TEXTLIST ErrorList
  0 = 'Minden rendben.'
  1 = 'Termék csatlakozó fedél\nnincs nyitva.'
  2 = 'Termék csatlakozó fedél\nnyitva van.'
  3 = 'Fütötömb hömérséklete\nnem megfelelö.'
  4 = 'Fütötömb hömérséklete\nmegfelelö.'
  5 = 'Sürített levegö nyomása\nnincs rendben.'
  6 = 'Sürített levegö nem kapcsolt ki.'
  7 = 'Nincs hegesztö\nelöfigyelmeztetés.'
  8 = 'Hegesztö\nelöfigyelmeztetés!'
  9 = 'Nem kell hegesztö elektródát\ncserélni.'
  10 = 'Hegesztö elektródát\nkell cserélni.'
  11 = 'A hegesztö még nem\nindult be.'
  12 = 'A hegesztö beindult.'
  13 = 'Nincs hegesztö áramhiba.'
  14 = 'Hegesztö áramhiba!'
  15 = 'Árammal hegesztés\nkikapcsolva!'
  16 = 'Árammal hegesztés\nbekapcsolva!'
  17 = 'A hegesztö nem üzemkész!'
  18 = 'A hegesztö üzemkész!'
  19 = 'NTC vágó: sebesség\nnem nulla.'
  20 = 'NTC vágó: sebesség nulla.'
  21 = 'NTC vágó: a sebesség\nnem állt be!'
  22 = 'NTC vágó: a sebesség\nbeállt!'
  23 = 'NTC vágó: nincs vészjelzés.'
  24 = 'NTC vágó: vészjelzés!'
  25 = 'NTC vágó: nem üzemkész!'
  26 = 'NTC vágó: üzemkész.'
  27 = 'Hegesztö: hegesztési\nfolyamat nincs kész.'
  28 = 'Hegesztö: hegesztési\nfolyamat kész.'
  29 = 'Pt oldali fénysorompó\nblokkolva.'
  30 = 'Pt oldali fénysorompó\nszabad.'
  31 = 'NTC oldali fénysorompó\nblokkolva.'
  32 = 'NTC oldali fénysorompó\nszabad.'
  33 = 'A kamera dolgozik.'
  34 = 'A kamera nem dolgozik.'
  35 = 'Kamera: a termék nincs jól\nrögzitve.'
  36 = 'Kamera: a termék jól\nvan rögzitve.'
  37 = 'Kamera: vezeték színsorrend\nnincs rendben.'
  38 = 'Kamera: vezeték színsorrend\nrendben van.'
  39 = 'Kamera: vezeték szigetelés\nnincs rendben.'
  40 = 'Kamera: vezeték szigetelés\nrendben van.'
  41 = 'A biztonsági relé földje megvan.'
  42 = 'A biztonsági relé földje hiányzik.\nValamelyik ajtó nyitva van?'
  43 = 'A biztonsági relé tápja hiányzik.\nValamelyik ajtó nyitva van?'
  44 = 'A biztonsági relé tápja megvan.'
  65 = 'Adapterlefogó nincs\nteljesen visszahúzva.'
  66 = 'Adapterlefogó\nteljesen visszahúzva.'
  67 = 'Adapterlefogó nem\naktiválódott.'
  68 = 'Az adapterlefogó aktív.'
  69 = 'Nem érzékel adaptert\na szánon!'
  70 = 'Fent van az adapter a szánon.'
  71 = 'A 3-as hegesztöfej nincs fent.'
  72 = 'A 3-as hegesztöfej fent van.'
  73 = 'A 3-as hegesztöfej nincs lent.'
  74 = 'A 3-as hegesztöfej lent van.'
  75 = 'A Pt oldali tengely plusz\nvégállásban van.'
  76 = 'A Pt oldali tengely nincs\nplusz \nvégállásban.'
  81 = 'Fütötömb nincs fent.'
  82 = 'Fütötömb fent van.'
  83 = 'Fütötömb nincs lent.'
  84 = 'Fütötömb lent van.'
  85 = 'Mérötük nincsenek kitolva.'
  86 = 'Mérötük ki vannak tolva.'
  87 = 'Mérötük nincsenek behúzva.'
  88 = 'Mérötük be vannak húzva.'
  89 = 'Lézer blende nincs bezárva.'
  90 = 'Lézer blende be van zárva.'
  91 = 'Lézer blende nincs kinyitva.'
  92 = 'Lézer blende ki van nyitva.'
  93 = 'Kappe prés legalul van.'
  94 = 'Kappe prés nincs legalul.'
  95 = 'A Pt oldali tengely minusz\nvégállásban van.'
  96 = 'A Pt oldali tengely nincs\nminusz \nvégállásban.'
  97 = 'Kappe prés jobb oldala\nnincs lent.'
  98 = 'Kappe prés jobb oldala\nlent van.'
  99 = 'Kappe prés jobb oldala\nnincs fent.'
  100 = 'Kappe prés jobb oldala\nfent van.'
  101 = 'Kappe prés bal oldala\nnincs fent.'
  102 = 'Kappe prés bal oldala\nfent van.'
  103 = 'Kappe prés bal oldala\nnincs lent.'
  104 = 'Kappe prés bal oldala\nlent van.'
  105 = 'A fütötömb nincs a szán\nfölött.'
  106 = 'A fütötömb a szán \nfölött van.'
  107 = 'A szigetelés mérötük\nnincsenek a szán fölött.'
  108 = 'A szigetelés mérötük\na szán fölött vannak.'
  109 = 'A kappe prés nincs fent.'
  110 = 'A kappe prés fent van.'
  111 = 'A nagyfeszültségü mérötü\nnincs lent.'
  112 = 'A nagyfeszültségü mérötü\nlent van.'
  113 = 'NTC vágó: vágó-hajlító\nnincs lent.'
  114 = 'NTC vágó: vágó-hajlító\nlent van.'
  115 = 'NTC vágó: vágó-hajlító\nnincs fent.'
  116 = 'NTC vágó: vágó-hajlító\nfent van.'
  117 = '2. hegesztö fej: Felsö elektróda\nnincs kitolva.'
  118 = '2. hegesztö fej: Felsö elektróda\nki van tolva.'
  119 = '2. hegesztö fej: Felsö elektróda\nnincs behúzva.'
  120 = '2. hegesztö fej: Felsö elektróda\nbe van húzva.'
  121 = '2. hegesztö fej: Alsó elektróda\nnincs behúzva.'
  122 = '2. hegesztö fej: Alsó elektróda\nbe van húzva.'
  123 = '2. hegesztö fej: Alsó elektróda\nnincs kitolva.'
  124 = '2. hegesztö fej: Alsó elektróda\nki van tolva.'
  125 = 'NTC oldali tengely minusz\nvégállásban van.'
  126 = 'NTC oldali tengely nincs\nminusz \nvégállásban.'
  127 = 'NTC vágó: az NTC nincs\nmegfelelö pozícióban.'
  128 = 'NTC vágó: az NTC\nmegfelelö pozícióban van.'
  129 = 'NTC vágó: NTC megfogó\nnincs nyitva.'
  130 = 'NTC vágó: NTC megfogó\nnyitva van.'
  131 = 'NTC vágó: NTC megfogó\nnincs zárva.'
  132 = 'NTC vágó: NTC megfogó\nzárva van.'
  133 = 'NTC vágó: NTC kiszedö\nnincs kitolva.'
  134 = 'NTC vágó: NTC kiszedö\nki van tolva.'
  135 = 'NTC vágó: NTC kiszedö\nnincs behúzva.'
  136 = 'NTC vágó: NTC kiszedö\nbe van húzva.'
  137 = 'NTC vágó: piros gomb\nnincs benyomva.'
  138 = 'NTC vágó: piros gomb\nbe van nyomva.'
  139 = 'NTC vágó: zöld gomb\nnincs benyomva.'
  140 = 'NTC vágó: zöld gomb\nbe van nyomva.'
  141 = 'Nincs megfelelö vágott NTC.'
  142 = 'Van vágott NTC.'
  145 = 'Elöhajlító: felsö pofa nincs lent.'
  146 = 'Elöhajlító: felsö pofa lent van.'
  147 = 'Elöhajlító: felsö pofa nincs fent.'
  148 = 'Elöhajlító: felsö pofa fent van.'
  149 = 'Elöhajlító: alsó pofa nincs lent.'
  150 = 'Elöhajlító: alsó pofa lent van.'
  151 = 'Elöhajlító: alsó pofa nincs fent.'
  152 = 'Elöhajlító: alsó pofa fent van.'
  153 = '1. hegesztöfej: bal elektróda\nnincs fent.'
  154 = '1. hegesztöfej: bal elektróda\nfent van.'
  155 = '1. hegesztöfej: bal elektróda\nnincs lent.'
  156 = '1. hegesztöfej: bal elektróda\nlent van.'
  161 = 'Véghajlító: felsö pofa nincs lent.'
  162 = 'Véghajlító: felsö pofa lent van.'
  163 = 'Véghajlító: felsö pofa nincs fent.'
  164 = 'Véghajlító: felsö pofa fent van.'
  165 = 'Véghajlító: alsó pofa nincs fent.'
  166 = 'Véghajlító: alsó pofa fent van.'
  167 = 'Véghajlító: alsó pofa nincs lent.'
  168 = 'Elöhajlító: alsó pofa lent van.'
  169 = '1. hegesztöfej: jobb elektróda\nnincs fent.'
  170 = '1. hegesztöfej: jobb elektróda\nfent van.'
  171 = '1. hegesztöfej: jobb elektróda\nnincs lent.'
  172 = '1. hegesztöfej: jobb elektróda\nlent van.'
  175 = 'NTC oldali tengely plusz\nvégállásban van.'
  176 = 'NTC oldali tengely nincs\nplusz végállásban.'
  193 = 'NTC oldali tengely nem\nüzemkész.'
  194 = 'NTC oldali tengely\nüzemkész.'
  195 = 'Pt oldali tengely nem\nüzemkész.'
  196 = 'Pt oldali tengely\nüzemkész.'
  197 = 'Nem kapcsolt be a\nnagyfeszültség.'
  198 = 'Nem kapcsolt ki a\nnagyfeszültség.'
  199 = 'Nincs a \nnagyfeszültség\na kappén.'
  200 = 'Rajta van a nagyfeszültség\na kappén.'
  201 = 'Nincs 48V a sokkoláshoz.'
  202 = 'Van 48V a sokkoláshoz.'
  203 = 'Nem kapcsolt ki a\nnagyfeszültség'
  204 = 'Kikapcsolt a nagyfeszültség.'
  205 = 'A Kappe prés nincs fent.'
  300 = 'NTC vágó állapothiba.'
  301 = 'NTC nem érkezett meg a\nvágáshoz.'
  302 = 'A robot a szán útjában lehet.'
  303 = 'A hegesztöt lefoglalta az\nNTC oldal.'
  304 = 'A hegesztöt lefoglalta a\nPt oldal.'
  305 = 'A robotot lefoglalta az\nNTC oldal.'
  306 = 'A robotot lefoglalta a\nPt oldal.'
  307 = 'A robotmüvelet elakadt.'
  308 = 'Kameramüvelet elakadt.'
  309 = 'Igazítsa meg/tegye fel a Pt pozícionáló\nfedelet, majd nyomja meg a\n"Tovább" gombot!'
  310 = 'Helyezzen be a helyére egy kappét,\nmajd nyomja meg a "Tovább" gombot!'
  311 = 'Nem sikerült a log fájlt\n megnyitni,\nvagy a mappáját létrehozni.'
  312 = 'Nem sikerült lekérdezni a\nlog fájl tulajdonságait.'
  313 = 'Nem sikerült a rendszeridöt\nlekérdezni.'
  314 = 'Nem sikerült írni a log fájlt.'
  315 = 'Nem sikerült a log fájl zárása.'
  316 = 'Nem sikerült létrehozni a log\nfájlnak a megfelelö mappát.'
  317 = 'Nincs lezárva a csatlakozó fedél.\nZárja le és nyomja meg a "Tovább"\ngombot!'
  318 = 'Hibás termék! Nyomja meg a\n"Tovább" gombot, és tegye a \nterméket a megfelelö helyre!'
  319 = 'Termékrögzítés, vezetéksorrend,\nhüvelyek rendben vannak?\nHa igen, nyomja meg a "Tovább" gombot!'
  320 = '1. hegesztés: alkatrész felismerési hiba!'
  321 = '3. hegesztés: alkatrész felismerési hiba!'
  322 = '2. hegesztés: alkatrész felismerési hiba!'
  323 = '4. hegesztés: alkatrész felismerési hiba!'
  324 = '5. hegesztés: alkatrész felismerési hiba!'
  325 = '1. hegesztés: a hegesztés nem megfelelő!'
  326 = '3. hegesztés: a hegesztés nem megfelelő!'
  327 = '2. hegesztés: a hegesztés nem megfelelő!'
  328 = '4. hegesztés: a hegesztés nem megfelelő!'
  329 = '5. hegesztés: a hegesztés nem megfelelő!'
  330 = '1. hegesztés: hegesztési hibát \njelzett a hegesztö'
  331 = '3. hegesztés: hegesztési hibát \njelzett a hegesztö'
  332 = '2. hegesztés: hegesztési hibát \njelzett a hegesztö'
  333 = '4. hegesztés: hegesztési hibát \njelzett a hegesztö'
  334 = '5. hegesztés: hegesztési hibát \njelzett a hegesztö'
  335 = '6. hegesztés: hegesztési hibát \njelzett a hegesztö'
  336 = '7. hegesztés: hegesztési hibát \njelzett a hegesztö'
  337 = 'Ellenörizze a hegesztést, vegye le\na Pt pozícionáló fedelet, majd nyomja\nmeg a "Tovább" gombot!'
  338 = 'Himba nincs elöl'
  339 = 'Himba nincs hátul'
  340 = 'Pt Kamera komm. kapcsolat nyitási hiba!'
  341 = 'Pt Kamera komm. küldési hiba!'
  342 = 'Pt Kamera komm. fogadási hiba!'
  343 = 'Pt Kamera komm. kapcsolat bezárási hiba!'
  344 = 'Pt Kamera nem érzékel terméket!'
  345 = 'Pt Kamera nem érzékel se adaptert, se kappét!\nEllenőrizze a terméket!'
  346 = 'Nincs kiválasztva művelet!'
  347 = 'Pt Kamera adat üres!'
  348 = 'Pt Kamera trigger TimeOut!'
  299 = 'Nincs NTC a hegesztésnél!'
  298 = 'Robot nem OK! Nyissa ki, zárja be a biztonsági ajtót!'
  297 = 'NTC érzékelő hiba!'
   = ''
END_TEXTLIST

(* stored: Version 1.1.0.1, ProductVersion 3.1.4024.11
   TextList ErrorList: Id {c8d4feed-67e6-48ea-be1b-9cb77b3af509} *)
